FUNCTION_BLOCK GrippingMachine IMPLEMENTS IMachine
VAR_INPUT
END_VAR
VAR_OUTPUT
END_VAR
VAR
	Xts : XtsTrack;
	stateMachine : PMLStateMachine;
	gearMovers : ARRAY [1..10] OF GearMover;
	XtsMovers : ARRAY [1..10] OF IMover;
	igearMovers : ARRAY[1..10] OF IGearMover;
	i : INT;
	bInit : BOOL;
END_VAR

IF NOT bInit THEN
	FOR i := 1 TO 10 DO
		igearMovers[i] := gearMovers[i];
		XtsMovers[i] := gearMovers[i];
	END_FOR
	stateMachine.PMLCommand(Command := Tc3_PackML_V2.E_PMLState.ePMLState_Aborting);
	IF stateMachine.getState() = Tc3_PackML_V2.E_PMLState.ePMLState_Aborting THEN
		stateMachine.StateComplete();
		bInit := TRUE;
	END_IF
END_IF
stateMachine();
Xts(MoverArray := XtsMovers, StateMachine := stateMachine);
FOR i := 1 TO 10 DO
	gearMovers[i](XtsTrack := Xts, StateMachine := stateMachine, MoverArray := igearMovers);	
END_FOR

{warning 'add property implementation'}
PROPERTY PMLState : PackMLState
GET
END_GET
END_PROPERTY

END_FUNCTION_BLOCK

(* stored: Version 1.1.0.1, ProductVersion 3.1.4024.9
   POU GrippingMachine: Id {cef35bf0-d94b-4472-a52e-67d847177915}, SpecialFunc None
   Property PMLState: Id {937222a3-3d9b-4063-a98b-bc4aad01a053}
   Get Get: Id {f520911b-40aa-4fe6-9082-3c0f7e93d822} *)
